{attribute 'GeneratedUsingTerminal: EL2521-0000-1017'}
{attribute addProperty BoxType "EL2521-0000-1017"}
{attribute addProperty Id "Set_counter_doneBOOL1Counter_underflowBOOL1Counter_overflowBOOL1Sync_ErrorBOOL1TxPDO_ToggleBOOL1"}
{attribute addProperty CRC "1863314867"}
{attribute addProperty Size "5"}
TYPE Status_6F0FEDB3 :
STRUCT
	{attribute addProperty Name "Set_counter_done"}
	Set_counter_done : BOOL;
	{attribute addProperty Name "Counter_underflow"}
	Counter_underflow : BOOL;
	{attribute addProperty Name "Counter_overflow"}
	Counter_overflow : BOOL;
	{attribute addProperty Name "Sync_Error"}
	Sync_Error : BOOL;
	{attribute addProperty Name "TxPDO_Toggle"}
	TxPDO_Toggle : BOOL;
END_STRUCT
END_TYPE

(* stored: Version 1.2.0.0, ProductVersion 3.1.4024.9
   DUT Status_6F0FEDB3: Id {b3f3aa75-4af3-4c7b-8e88-9186bc60b6e4} *)
